{attribute 'qualified_only'}
{attribute 'strict'}
TYPE E_ProcessCylinder_State :
(
		//GENERIC
	ABORTED				,
	HOMING				,
	READY				,
	MANUAL_MODE			,
	STOPPING			,
	//SPECIFIC FOR EVERY STATION
	EXTEND_PROCESS_CYLINDER,
	RETRACT_PROCESS_CYLINDER,
	DONE				,
	RESET				
);
END_TYPE

(* stored: Version 1.1.0.1, ProductVersion 3.1.4024.13
   DUT E_ProcessCylinder_State: Id {39ea7c49-57ae-4672-9d34-1fe246bace50} *)
